TYPE U_SAFETY_ESTOP :
UNION
	stStatusWords					: ST_SAFETY_FBStatus;		(* BUnknown, BState, wDiagnosis, wInputs, wOutputs - takie same dla wszystkich FB *)
	stStatus						: ST_SAFETY_ESTOP; 			(* Rozbite na Bity - inne dla kazdego bloku*)
END_UNION
END_TYPE

(* stored: Version 1.1.0.1, ProductVersion 3.1.4022.12
   DUT U_SAFETY_ESTOP: Id {a839d9e7-58b1-4501-bbc7-3016ec5d920f} *)
